// TIA Portal V19 export
FUNCTION "DecoilersHRot_CALL" : Void   // FC126, LAD
TITLE = DECOILERS HORIZONTAL ROTATION & TRANSLATION CALL
// stored: SetENOAutomatically false
BEGIN

REGION Network 1 (SCL): DataIn
   // Gen
   "DecoilersHRot".DataIn.PB_Decoiler1_MoveInLine := "A01_HMI".MB1.Button.CoilHandling.DecoilersHRot.Move_InLineDecoiler1 OR "LB101".PB.Decoiler1InLine;
   "DecoilersHRot".DataIn.PB_Decoiler2_MoveInLine := "A01_HMI".MB1.Button.CoilHandling.DecoilersHRot.Move_InLineDecoiler2 OR "LB101".PB.Decoiler2InLine;


   // Rotation
   "DecoilersHRot".DataIn.Rotation.PB := "A01_HMI".MB1.Button.CoilHandling.DecoilersHRot.Rotation;

   "DecoilersHRot".DataIn.Rotation.Rest_Ls[1] := "D02_Ls";
   "DecoilersHRot".DataIn.Rotation.Work_Ls[1] := "D03_Ls";

   //Pivot
   "DecoilersHRot".DataIn.Pivot.PB := "A01_HMI".MB1.Button.CoilHandling.DecoilersHRot.Pivot;

   "DecoilersHRot".DataIn.Pivot.Rest_Ls[1] := "DecoilersHRot_Pivot_Ls_Rest";
   "DecoilersHRot".DataIn.Pivot.Work_Ls[1] := "DecoilersHRot_Pivot_Ls_Work";


   //Traslation
   "DecoilersHRot".DataIn.Traslation.PB := "A01_HMI".MB1.Button.CoilHandling.DecoilersHRot.Translation;

   "DecoilersHRot".DataIn.Traslation.LS_Minus :=
   "DecoilersHRot".DataIn.Traslation.LS_Plus :=
   "DecoilersHRot".DataIn.Traslation.Fan_M_ThermalProtection :=
   "DecoilersHRot".DataIn.Traslation.Fan_M_Feedback :=
   "DecoilersHRot".DataIn.Traslation.Brake_M_Q :=
   "DecoilersHRot".DataIn.Traslation.Brake_M_Feedback := "Sys".ByPass;
END_REGION

REGION Network 2: >
END_REGION

REGION Network 3 (SCL): CIn - Manager
   "DecoilersHRot".CIn.Manager := "CoilHandling".COut.DecoilersHRot;

   "DecoilersHRot".CIn.CoilCar_OutOfLine := "Coilcar".COut.IsOutline;
END_REGION

REGION Network 4: CIn - Pressure running
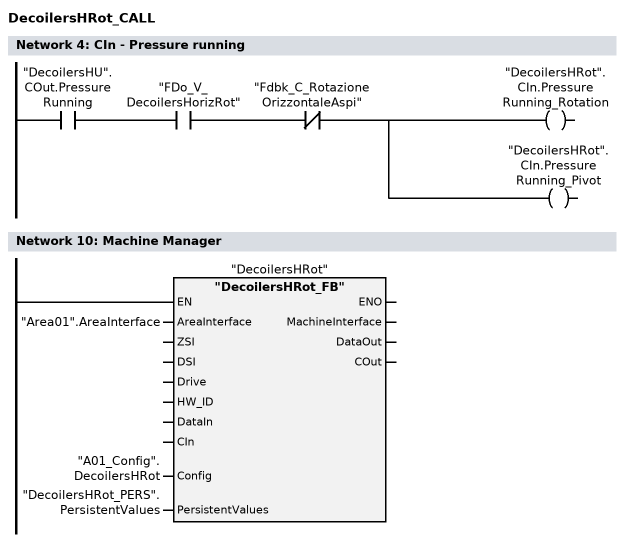
   RUNG wire#powerrail
      Contact( "DecoilersHU".COut.PressureRunning )
      Contact( "FDo_V_DecoilersHorizRot" )
      I_Contact( "Fdbk_C_RotazioneOrizzontaleAspi" )
      wire#w1
      Coil( "DecoilersHRot".CIn.PressureRunning_Rotation )
   END_RUNG
   RUNG wire#w1
      Coil( "DecoilersHRot".CIn.PressureRunning_Pivot )
   END_RUNG
   // the same network as SCL:
   "DecoilersHRot".CIn.PressureRunning_Rotation := "DecoilersHU".COut.PressureRunning AND "FDo_V_DecoilersHorizRot" AND NOT "Fdbk_C_RotazioneOrizzontaleAspi";
   "DecoilersHRot".CIn.PressureRunning_Pivot := "DecoilersHRot".CIn.PressureRunning_Rotation;
END_REGION

REGION Network 5: >
END_REGION

REGION Network 6 (SCL): DSI
   "DecoilersHRot".DSI.Translation := "F_DB".DSI_S120_DecoilersTranslation;
   "DecoilersHRot".DSI.Rotation :=
   "DecoilersHRot".DSI.Pivot := "F_DB".DSI_V_DecoilersHorizRotation;
END_REGION

REGION Network 7 (SCL): Drive
   "DecoilersHRot".Drive.Traslation.Infeed_ON := "Areas_ITF".AG.Infeed_Running;
   "DecoilersHRot".Drive.Traslation.AccessPoint := "HW_Const_Values".CU1_PN_690A1_1_ModuleAccessPoint;
   "DecoilersHRot".Drive.Traslation.AxisID := "CU1_ID_5_690A1_1_690M1";
   "DecoilersHRot".Drive.Traslation.TokenChain := "TOKENCHAIN_CU1";
END_REGION

REGION Network 8 (SCL): HW ID
   "DecoilersHRot".HW_ID.Traslation_TEL1 := "HW_Const_Values".CU1_PN_690A1_1_Standard_telegram_1;
   "DecoilersHRot".HW_ID.TraslationEnc_IO := "HW_Const_Values".HW_694P1_Telegram_81_DI_DO;
END_REGION

REGION Network 9: >
END_REGION

REGION Network 10: Machine Manager
   RUNG wire#powerrail
      "DecoilersHRot"(AreaInterface := "Area01".AreaInterface, ZSI :=, DSI :=, Drive :=, HW_ID :=, DataIn :=, CIn :=, Config := "A01_Config".DecoilersHRot, PersistentValues := "DecoilersHRot_PERS".PersistentValues, MachineInterface =>, DataOut =>, COut =>)
   END_RUNG
   // the same network as SCL:
   "DecoilersHRot"(AreaInterface := "Area01".AreaInterface,   // "DecoilersHRot_FB"
                   Config := "A01_Config".DecoilersHRot,
                   PersistentValues := "DecoilersHRot_PERS".PersistentValues);
END_REGION

REGION Network 11: >
END_REGION

REGION Network 12 (SCL): Data Out
   //Gen
   (*
   "DecoilersHRot_TowerLamp_SL102" := "DecoilersHRot".DataOut.Tower_Lamp;
   "DecoilersHRot_TowerHorn_SL102" := "DecoilersHRot".DataOut.Tower_Horn;
   *)

   //Rotation
   "DecoilersHRot_Rotation_V_Dec1InLine" := "DecoilersHRot".DataOut.Rotation.RestSolenoid;
   "DecoilersHRot_Rotation_V_Dec2InLine" := "DecoilersHRot".DataOut.Rotation.WorkSolenoid;

   //Pivot
   "DecoilersHRot_Pivot_V_Rest" := "DecoilersHRot".Pivot.V.RestSolenoid;
   "DecoilersHRot_Pivot_V_Work" := "DecoilersHRot".Pivot.V.WorkSolenoid;
END_REGION

REGION Network 13: >
END_REGION

REGION Network 14: >
END_REGION

REGION Network 15: >
END_REGION
END_FUNCTION
